Fanuc TP program (LS listing): _init_pos.ls

/PROG  _INIT_POS
/ATTR
OWNER		= MNEDITOR;
COMMENT		= "Init Positions";
PROG_SIZE	= 273;
CREATE		= DATE 22-12-15  TIME 10:15:36;
MODIFIED	= DATE 24-12-02  TIME 13:42:28;
FILE_NAME	= ;
VERSION		= 0;
LINE_COUNT	= 7;
MEMORY_SIZE	= 749;
PROTECT		= READ_WRITE;
TCD:  STACK_SIZE	= 0,
      TASK_PRIORITY	= 50,
      TIME_SLICE	= 0,
      BUSY_LAMP_OFF	= 0,
      ABORT_REQUEST	= 0,
      PAUSE_REQUEST	= 0;
DEFAULT_GROUP	= 1,*,*,*,*;
CONTROL_CODE	= 00000000 00000000;
LOCAL_REGISTERS	= 0,0,0;
/APPL

AUTO_SINGULARITY_HEADER;
  ENABLE_SINGULARITY_AVOIDANCE   : TRUE;
/MN
   1:  !*********INIT ROBOT POS********* ;
   2:  LBL[100] ;
   3:  DO[42:OFF:At Outfd Recon]=OFF ;
   4:  JMP LBL[999] ;
   5:   ;
   6:   ;
   7:  LBL[999] ;
/POS
/END
